# EPICS autosave request: iocs/mmpadIOC/iocBoot/iocMMPAD/auto_settings.req
file "mmpad_settings.req",        P=$(P),  R=cam1:
file "NDStdArrays_settings.req",  P=$(P),  R=image1:
file "commonPlugin_settings.req", P=$(P)
